Staubli VAL3: VelocityType.pjx

--- VelocityType.pjx ---
Parameters version=s7.8.1 stackSize=5000 millimeterUnit=true
Program file=start.pgx
Program file=stop.pgx
Data file=VelocityType.dtx

--- VelocityType.dtx ---
public num INVALID
public num JOINT
public num BASE_FRAME
public num TOOL_FRAME
